// TIA Portal V19 export
FUNCTION "FC80_Greasing" : Void   // FC80, LAD
{ S7_Optimized_Access := 'TRUE' }
// stored: AutoNumber false, SetENOAutomatically false
BEGIN

REGION Network 1: Manage greasing X axis
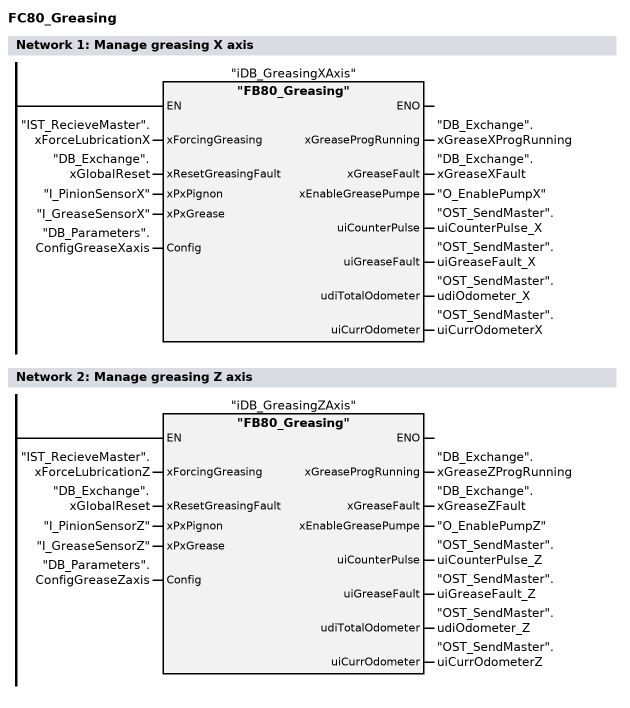
   RUNG wire#powerrail
      "iDB_GreasingXAxis"(xForcingGreasing := "IST_RecieveMaster".xForceLubricationX, xResetGreasingFault := "DB_Exchange".xGlobalReset, xPxPignon := "I_PinionSensorX", xPxGrease := "I_GreaseSensorX", Config := "DB_Parameters".ConfigGreaseXaxis, xGreaseProgRunning => "DB_Exchange".xGreaseXProgRunning, xGreaseFault => "DB_Exchange".xGreaseXFault, xEnableGreasePumpe => "O_EnablePumpX", uiCounterPulse => "OST_SendMaster".uiCounterPulse_X, uiGreaseFault => "OST_SendMaster".uiGreaseFault_X, udiTotalOdometer => "OST_SendMaster".udiOdometer_X, uiCurrOdometer => "OST_SendMaster".uiCurrOdometerX)
   END_RUNG
   // the same network as SCL:
   "iDB_GreasingXAxis"(xForcingGreasing := "IST_RecieveMaster".xForceLubricationX,   // "FB80_Greasing"
                       xResetGreasingFault := "DB_Exchange".xGlobalReset,
                       xPxPignon := "I_PinionSensorX",
                       xPxGrease := "I_GreaseSensorX",
                       Config := "DB_Parameters".ConfigGreaseXaxis,
                       xGreaseProgRunning => "DB_Exchange".xGreaseXProgRunning,
                       xGreaseFault => "DB_Exchange".xGreaseXFault,
                       xEnableGreasePumpe => "O_EnablePumpX",
                       uiCounterPulse => "OST_SendMaster".uiCounterPulse_X,
                       uiGreaseFault => "OST_SendMaster".uiGreaseFault_X,
                       udiTotalOdometer => "OST_SendMaster".udiOdometer_X,
                       uiCurrOdometer => "OST_SendMaster".uiCurrOdometerX);
END_REGION

REGION Network 2: Manage greasing Z axis
   RUNG wire#powerrail
      "iDB_GreasingZAxis"(xForcingGreasing := "IST_RecieveMaster".xForceLubricationZ, xResetGreasingFault := "DB_Exchange".xGlobalReset, xPxPignon := "I_PinionSensorZ", xPxGrease := "I_GreaseSensorZ", Config := "DB_Parameters".ConfigGreaseZaxis, xGreaseProgRunning => "DB_Exchange".xGreaseZProgRunning, xGreaseFault => "DB_Exchange".xGreaseZFault, xEnableGreasePumpe => "O_EnablePumpZ", uiCounterPulse => "OST_SendMaster".uiCounterPulse_Z, uiGreaseFault => "OST_SendMaster".uiGreaseFault_Z, udiTotalOdometer => "OST_SendMaster".udiOdometer_Z, uiCurrOdometer => "OST_SendMaster".uiCurrOdometerZ)
   END_RUNG
   // the same network as SCL:
   "iDB_GreasingZAxis"(xForcingGreasing := "IST_RecieveMaster".xForceLubricationZ,   // "FB80_Greasing"
                       xResetGreasingFault := "DB_Exchange".xGlobalReset,
                       xPxPignon := "I_PinionSensorZ",
                       xPxGrease := "I_GreaseSensorZ",
                       Config := "DB_Parameters".ConfigGreaseZaxis,
                       xGreaseProgRunning => "DB_Exchange".xGreaseZProgRunning,
                       xGreaseFault => "DB_Exchange".xGreaseZFault,
                       xEnableGreasePumpe => "O_EnablePumpZ",
                       uiCounterPulse => "OST_SendMaster".uiCounterPulse_Z,
                       uiGreaseFault => "OST_SendMaster".uiGreaseFault_Z,
                       udiTotalOdometer => "OST_SendMaster".udiOdometer_Z,
                       uiCurrOdometer => "OST_SendMaster".uiCurrOdometerZ);
END_REGION
END_FUNCTION
